FUNCTION_BLOCK OR_NOT (* Composite Function Block Type *)
  (* Standard: 61499-2 *)
  (* Version 0.0, 7/11/2026, Schneider Electric, template *)
  PACKAGE SE.Nereda;
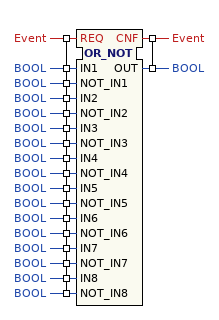
  EVENT_INPUT
    REQ WITH IN1, NOT_IN1, IN2, NOT_IN2, IN3, NOT_IN3, IN4, NOT_IN4, IN5, NOT_IN5, IN6, NOT_IN6, IN7, NOT_IN7, IN8, NOT_IN8; (* Normal Execution Request *)
  END_EVENT
  EVENT_OUTPUT
    CNF WITH OUT; (* Input changed *)
  END_EVENT
  VAR_INPUT
    IN1 : BOOL; (* Argument *)
    NOT_IN1 : BOOL; (* Argument *)
    IN2 : BOOL; (* Argument *)
    NOT_IN2 : BOOL; (* Argument *)
    IN3 : BOOL; (* Argument *)
    NOT_IN3 : BOOL; (* Argument *)
    IN4 : BOOL; (* Argument *)
    NOT_IN4 : BOOL; (* Argument *)
    IN5 : BOOL; (* Argument *)
    NOT_IN5 : BOOL; (* Argument *)
    IN6 : BOOL; (* Argument *)
    NOT_IN6 : BOOL; (* Argument *)
    IN7 : BOOL; (* Argument *)
    NOT_IN7 : BOOL; (* Argument *)
    IN8 : BOOL; (* Argument *)
    NOT_IN8 : BOOL; (* Argument *)
  END_VAR
  VAR_OUTPUT
    OUT : BOOL; (* Output value *)
  END_VAR
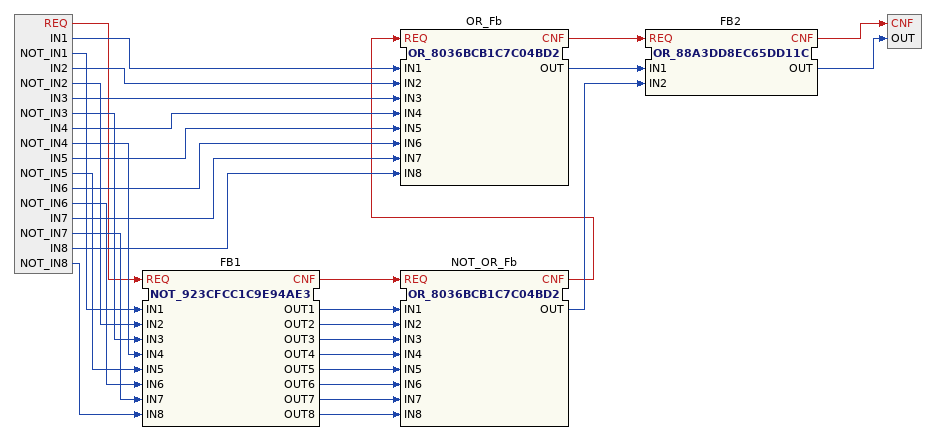
  FBS
    OR_Fb : OR_8036BCB1C7C04BD2; {SET_ATTRIBUTE(Configuration.GenericFBType.InterfaceParams, Runtime.Standard#CNT:=8;OUT:BOOL)}
    FB1 : NOT_923CFCC1C9E94AE3; {SET_ATTRIBUTE(Configuration.GenericFBType.InterfaceParams, Runtime.Standard#CNT:=8;OUT${CNT$}:BOOL,BOOL,BOOL,BOOL,BOOL,BOOL,BOOL,BOOL)}
    NOT_OR_Fb : OR_8036BCB1C7C04BD2; {SET_ATTRIBUTE(Configuration.GenericFBType.InterfaceParams, Runtime.Standard#CNT:=8;OUT:BOOL)}
    FB2 : OR_88A3DD8EC65DD11C; {SET_ATTRIBUTE(Configuration.GenericFBType.InterfaceParams, Runtime.Standard#CNT:=2;OUT:BOOL)}
  END_FBS
  EVENT_CONNECTIONS
    OR_Fb.CNF TO FB2.REQ;
    FB1.CNF TO NOT_OR_Fb.REQ;
    NOT_OR_Fb.CNF TO OR_Fb.REQ;
    REQ TO FB1.REQ;
    FB2.CNF TO CNF;
  END_CONNECTIONS
  DATA_CONNECTIONS
    OR_Fb.OUT TO FB2.IN1;
    IN1 TO OR_Fb.IN1;
    NOT_IN1 TO FB1.IN1;
    IN2 TO OR_Fb.IN2;
    NOT_IN2 TO FB1.IN2;
    IN3 TO OR_Fb.IN3;
    NOT_IN3 TO FB1.IN3;
    IN4 TO OR_Fb.IN4;
    NOT_IN4 TO FB1.IN4;
    IN5 TO OR_Fb.IN5;
    NOT_IN5 TO FB1.IN5;
    IN6 TO OR_Fb.IN6;
    NOT_IN6 TO FB1.IN6;
    IN7 TO OR_Fb.IN7;
    NOT_IN7 TO FB1.IN7;
    IN8 TO OR_Fb.IN8;
    NOT_IN8 TO FB1.IN8;
    FB1.OUT1 TO NOT_OR_Fb.IN1;
    FB1.OUT2 TO NOT_OR_Fb.IN2;
    FB1.OUT3 TO NOT_OR_Fb.IN3;
    FB1.OUT4 TO NOT_OR_Fb.IN4;
    FB1.OUT5 TO NOT_OR_Fb.IN5;
    FB1.OUT6 TO NOT_OR_Fb.IN6;
    FB1.OUT7 TO NOT_OR_Fb.IN7;
    FB1.OUT8 TO NOT_OR_Fb.IN8;
    NOT_OR_Fb.OUT TO FB2.IN2;
    FB2.OUT TO OUT;
  END_CONNECTIONS
END_FUNCTION_BLOCK
